Staubli VAL3: movingReporter.pgx

program movingReporter()
  local bool settled
begin
  settled = false

  while true
    wait(isSettled() != settled)
    settled = !settled

    call sendMoving()
  endWhile
end
